FUNCTION_BLOCK INTERNAL FINAL POU_2
VAR_INPUT
END_VAR
VAR_OUTPUT
END_VAR
VAR
END_VAR

END_FUNCTION_BLOCK

(* stored: Version 1.1.0.1, ProductVersion 3.1.4024.12
   POU POU_2: Id {c15b4ad9-2bb9-41e7-9596-f650694ee921}, SpecialFunc None *)
